{attribute 'GeneratedUsingTerminal: EL3318-0000-0016'}
{attribute addProperty BoxType "EL3318-0000-0016"}
{attribute addProperty Id "StatusAT %I*Status_68C33E995ValueAT %I*INT2"}
{attribute addProperty CRC "2507538081"}
{attribute addProperty Size "7"}
TYPE TC_Channel_9575FEA1 :
STRUCT
	{attribute addProperty Name "Status"}
	Status AT %I* : Status_68C33E99;
	{attribute addProperty Name "Value"}
	Value AT %I* : INT;
END_STRUCT
END_TYPE

(* stored: Version 1.2.0.0, ProductVersion 3.1.4024.9
   DUT TC_Channel_9575FEA1: Id {be34520d-9291-4925-9ead-56e271afa973} *)
